DATA_BLOCK "Db Plc <=> HMI"	// DB 100
TITLE = PLC <=> HMI EXCHANGED DATA
AUTHOR : Milesi
VERSION : 0.1
  STRUCT
   BUFFER_DATI : STRUCT
    BD1 : WORD ;	//Numero di ricetta corrente
    BD2 : WORD ;	//Numero di set di dati corrente
    BD3 : WORD ;	//Riservato
    BD4 : WORD ;	//Stato di tresferimento
    BD5 : WORD ;	//Riservato
   END_STRUCT ;
   BUFFER_ORDINI : STRUCT
    BO1 : WORD ;	//0 - Numero di ordine
    BO2 : WORD ;	//Parametro 1
    BO3 : WORD ;	//Parametro 2
    BO4 : WORD ;	//Parametro 3
   END_STRUCT ;
   BUFFER_PAGINE : STRUCT
    BP1 : WORD ;	//Tipo di pagina corrente
    BP2 : WORD ;	//Numero di pagina corrente
    BP3 : WORD ;	//Riservato
    BP4 : WORD ;	//Numero di campo corrente
    BP5 : WORD ;	//Riservato
   END_STRUCT ;
   DB100_DBW28 : WORD ;
   DB100_DBW30 : WORD ;
   DB100_DBW32 : WORD ;
   DB100_DBW34 : WORD ;
   DB100_DBW36 : WORD ;
   DB100_DBW38 : WORD ;
   DB100_DBW40 : WORD ;
   DB100_DBW42 : WORD ;
   DB100_DBW44 : WORD ;
   DB100_DBW46 : WORD ;
   DB100_DBW48 : WORD ;
   DB100_DBW50 : WORD ;
   DB100_DBW52 : WORD ;
   DB100_DBW54 : WORD ;
   DB100_DBW56 : WORD ;
   DB100_DBW58 : WORD ;
   DB100_DBW60 : WORD ;
   DB100_DBW62 : WORD ;
   DB100_DBW64 : WORD ;
   DB100_DBW66 : WORD ;
   DB100_DBW68 : WORD ;
   DB100_DBW70 : WORD ;
   DB100_DBW72 : WORD ;
   DB100_DBW74 : WORD ;
   DB100_DBW76 : WORD ;
   DB100_DBW78 : WORD ;
   DB100_DBW80 : WORD ;
   DB100_DBW82 : WORD ;
   DB100_DBW84 : WORD ;
   DB100_DBW86 : WORD ;
   DB100_DBW88 : WORD ;
   DB100_DBW90 : WORD ;
   DB100_DBW92 : WORD ;
   DB100_DBW94 : WORD ;
   DB100_DBW96 : WORD ;
   DB100_DBW98 : WORD ;
   PROFIBUS : STRUCT
    DB100_DBX100_0 : BOOL ;	//009 Cage 18 motor drive profibus slave 9 fault
    DB100_DBX100_1 : BOOL ;	//010 Cage 12 preforming motor drive profibus slave 10 fault
    DB100_DBX100_2 : BOOL ;	//011 Cage 12 motor drive profibus slave 11 fault
    DB100_DBX100_3 : BOOL ;	//012 Cage 6 motor drive profibus slave 12 fault
    DB100_DBX100_4 : BOOL ;	//013 Take-up unit ET200S profibus slave 20 fault
    DB100_DBX100_5 : BOOL ;	//014 Cage 24 ET200M profibus slave 21 fault
    DB100_DBX100_6 : BOOL ;	//015 Cage 18 ET200M profibus slave 22 fault
    DB100_DBX100_7 : BOOL ;	//016 Cage 12 ET200M profibus slave 23 fault
    DB100_DBX101_0 : BOOL ;	//001 Take-up traverse motor drive profibus slave 3 fault
    DB100_DBX101_1 : BOOL ;	//002 Take-up bobbin motor drive profibus slave 4 fault
    DB100_DBX101_2 : BOOL ;	//003 Capstan motor drive profibus slave 5 fault
    DB100_DBX101_3 : BOOL ;	//004
    DB100_DBX101_4 : BOOL ;	//005
    DB100_DBX101_5 : BOOL ;	//006 Cage 24 preforming motor drive profibus slave 7 fault
    DB100_DBX101_6 : BOOL ;	//007 Cage 24 motor drive profibus slave 6 fault
    DB100_DBX101_7 : BOOL ;	//008 Cage 18 preforming motor drive profibus slave 8 fault
   END_STRUCT ;
   PROFIBUS_1 : STRUCT
    DB100_DBX102_0 : BOOL ;	//025
    DB100_DBX102_1 : BOOL ;	//026
    DB100_DBX102_2 : BOOL ;	//027
    DB100_DBX102_3 : BOOL ;	//028
    DB100_DBX102_4 : BOOL ;	//029
    DB100_DBX102_5 : BOOL ;	//030
    DB100_DBX102_6 : BOOL ;	//031
    DB100_DBX102_7 : BOOL ;	//032
    DB100_DBX103_0 : BOOL ;	//017 Cage 6 ET200M profibus slave 24 fault
    DB100_DBX103_1 : BOOL ;	//018 Pay-off unit ET200S profibus slave 25 fault
    DB100_DBX103_2 : BOOL ;	//019 Pay-off traverse motor drive profibus slave 13 fault
    DB100_DBX103_3 : BOOL ;	//020
    DB100_DBX103_4 : BOOL ;	//021
    DB100_DBX103_5 : BOOL ;	//022
    DB100_DBX103_6 : BOOL ;	//023
    DB100_DBX103_7 : BOOL ;	//024
   END_STRUCT ;
   TRAVERSE : STRUCT
    DB100_DBX104_0 : BOOL ;	//041
    DB100_DBX104_1 : BOOL ;	//042
    DB100_DBX104_2 : BOOL ;	//043
    DB100_DBX104_3 : BOOL ;	//044
    DB100_DBX104_4 : BOOL ;	//045
    DB100_DBX104_5 : BOOL ;	//046
    DB100_DBX104_6 : BOOL ;	//047
    DB100_DBX104_7 : BOOL ;	//048
    DB100_DBX105_0 : BOOL ;	//033 Take-up traverse driven pintle emergency alarm
    DB100_DBX105_1 : BOOL ;	//034 Take-up traverse idle pintle emergency alarm
    DB100_DBX105_2 : BOOL ;	//034 Take-up traverse motor blower overload
    DB100_DBX105_3 : BOOL ;	//036 Take-up traverse motor drive fault
    DB100_DBX105_4 : BOOL ;	//037
    DB100_DBX105_5 : BOOL ;	//038
    DB100_DBX105_6 : BOOL ;	//039
    DB100_DBX105_7 : BOOL ;	//040
   END_STRUCT ;
   TAKE_UP_1 : STRUCT
    DB100_DBX106_0 : BOOL ;	//057 Take-up bobbin down
    DB100_DBX106_1 : BOOL ;	//058 Take-up bobbin off
    DB100_DBX106_2 : BOOL ;	//059
    DB100_DBX106_3 : BOOL ;	//060
    DB100_DBX106_4 : BOOL ;	//061
    DB100_DBX106_5 : BOOL ;	//062
    DB100_DBX106_6 : BOOL ;	//063
    DB100_DBX106_7 : BOOL ;	//064
    DB100_DBX107_0 : BOOL ;	//049 Take-up 24VDC power supply overload
    DB100_DBX107_1 : BOOL ;	//050 Take-up 230VAC power supply overload
    DB100_DBX107_2 : BOOL ;	//051 Take-up AC motors overload
    DB100_DBX107_3 : BOOL ;	//052 Take-up bobbin motor blower overload
    DB100_DBX107_4 : BOOL ;	//053 Take-up bobbin motor electric brake overload
    DB100_DBX107_5 : BOOL ;	//054 Take-up bobbin motor overtemperature
    DB100_DBX107_6 : BOOL ;	//055 Take-up bobbin motor drive fault
    DB100_DBX107_7 : BOOL ;	//056 Take-up bobbin stop series push-button alarm
   END_STRUCT ;
   CAPSTAN : STRUCT
    DB100_DBX108_0 : BOOL ;	//073
    DB100_DBX108_1 : BOOL ;	//074
    DB100_DBX108_2 : BOOL ;	//075
    DB100_DBX108_3 : BOOL ;	//076
    DB100_DBX108_4 : BOOL ;	//077
    DB100_DBX108_5 : BOOL ;	//078
    DB100_DBX108_6 : BOOL ;	//079
    DB100_DBX108_7 : BOOL ;	//080
    DB100_DBX109_0 : BOOL ;	//065 Capstan motor blower overload
    DB100_DBX109_1 : BOOL ;	//066
    DB100_DBX109_2 : BOOL ;	//067 Capstan motor brake control alarm
    DB100_DBX109_3 : BOOL ;	//068 Capstan main air minimum pressure
    DB100_DBX109_4 : BOOL ;	//069 Cable block open alarm
    DB100_DBX109_5 : BOOL ;	//070 Cable block close after run alarm
    DB100_DBX109_6 : BOOL ;	//071 Capstan motor drive fault
    DB100_DBX109_7 : BOOL ;	//072 Capstan motor overtemperature
   END_STRUCT ;
   Spare : STRUCT
    DB100_DBX110_0 : BOOL ;	//089
    DB100_DBX110_1 : BOOL ;	//090
    DB100_DBX110_2 : BOOL ;	//091
    DB100_DBX110_3 : BOOL ;	//092
    DB100_DBX110_4 : BOOL ;	//093
    DB100_DBX110_5 : BOOL ;	//094
    DB100_DBX110_6 : BOOL ;	//095
    DB100_DBX110_7 : BOOL ;	//096
    DB100_DBX111_0 : BOOL ;	//081
    DB100_DBX111_1 : BOOL ;	//082
    DB100_DBX111_2 : BOOL ;	//083
    DB100_DBX111_3 : BOOL ;	//084
    DB100_DBX111_4 : BOOL ;	//085
    DB100_DBX111_5 : BOOL ;	//086
    DB100_DBX111_6 : BOOL ;	//087
    DB100_DBX111_7 : BOOL ;	//088
   END_STRUCT ;
   CAGE24_1 : STRUCT
    DB100_DBX112_00 : BOOL ;	//105 Cage 24 open front guard
    DB100_DBX112_01 : BOOL ;	//106 Cage 24 presence of man
    DB100_DBX112_02 : BOOL ;	//107 Cage 24 loading engaged
    DB100_DBX112_03 : BOOL ;	//108 Cage 24 loading gear box not engaged
    DB100_DBX112_04 : BOOL ;	//109 Cage 24 loading motor overload
    DB100_DBX112_05 : BOOL ;	//110 Cage 24 air pipe not in position
    DB100_DBX112_06 : BOOL ;	//111 Cage 24
    DB100_DBX112_07 : BOOL ;	//112 Cage 24 piston inside cage
    DB100_DBX113_00 : BOOL ;	//097 Cage 24 24VDC power supply overload
    DB100_DBX113_01 : BOOL ;	//098 Cage 24 230VAC power supply overload
    DB100_DBX113_02 : BOOL ;	//099 Cage 24 motor blower overload
    DB100_DBX113_03 : BOOL ;	//100 Cage 24
    DB100_DBX113_04 : BOOL ;	//101 Cage 24 loading platform overload
    DB100_DBX113_05 : BOOL ;	//102 Cage 24 guard blower motor overload
    DB100_DBX113_06 : BOOL ;	//103 Cage 24 open front door
    DB100_DBX113_07 : BOOL ;	//104 Cage 24 open rear door
   END_STRUCT ;
   CAGE24_2 : STRUCT
    DB100_DBX114_00 : BOOL ;	//121 Cage 24 bobbin 1 break of wire
    DB100_DBX114_01 : BOOL ;	//122 Cage 24 bobbin 2 break of wire
    DB100_DBX114_02 : BOOL ;	//123 Cage 24 bobbin 3 break of wire
    DB100_DBX114_03 : BOOL ;	//124 Cage 24 bobbin 4 break of wire
    DB100_DBX114_04 : BOOL ;	//125 Cage 24 bobbin 5 break of wire
    DB100_DBX114_05 : BOOL ;	//126 Cage 24 bobbin 6 break of wire
    DB100_DBX114_06 : BOOL ;	//127 Cage 24 bobbin 7 break of wire
    DB100_DBX114_07 : BOOL ;	//128 Cage 24 bobbin 8 break of wire
    DB100_DBX115_00 : BOOL ;	//113 Cage 24 bobbin 9 break of wire
    DB100_DBX115_01 : BOOL ;	//114 Cage 24 bobbin 10 break of wire
    DB100_DBX115_02 : BOOL ;	//115 Cage 24 bobbin 11 break of wire
    DB100_DBX115_03 : BOOL ;	//116 Cage 24 bobbin 12 break of wire
    DB100_DBX115_04 : BOOL ;	//117 Cage 24 bobbin 13 break of wire
    DB100_DBX115_05 : BOOL ;	//118 Cage 24 bobbin 14 break of wire
    DB100_DBX115_06 : BOOL ;	//119 Cage 24 bobbin 15 break of wire
    DB100_DBX115_07 : BOOL ;	//120 Cage 24 bobbin 16 break of wire
   END_STRUCT ;
   CAGE24_3 : STRUCT
    DB100_DBX116_00 : BOOL ;	//137 Cage 24 bobbin 17 break of wire
    DB100_DBX116_01 : BOOL ;	//138 Cage 24 bobbin 18 break of wire
    DB100_DBX116_02 : BOOL ;	//139 Cage 24 bobbin 19 break of wire
    DB100_DBX116_03 : BOOL ;	//140 Cage 24 bobbin 20 break of wire
    DB100_DBX116_04 : BOOL ;	//141 Cage 24 bobbin 21 break of wire
    DB100_DBX116_05 : BOOL ;	//142 Cage 24 bobbin 22 break of wire
    DB100_DBX116_06 : BOOL ;	//143 Cage 24 bobbin 23 break of wire
    DB100_DBX116_07 : BOOL ;	//144 Cage 24 bobbin 24 break of wire
    DB100_DBX117_00 : BOOL ;	//129
    DB100_DBX117_01 : BOOL ;	//130
    DB100_DBX117_02 : BOOL ;	//131
    DB100_DBX117_03 : BOOL ;	//132
    DB100_DBX117_04 : BOOL ;	//133
    DB100_DBX117_05 : BOOL ;	//134
    DB100_DBX117_06 : BOOL ;	//135 Cage 24 break wire from ring
    DB100_DBX117_07 : BOOL ;	//136 Cage 24 insert wire control alarm
   END_STRUCT ;
   CAGE24_4 : STRUCT
    DB100_DBX118_00 : BOOL ;	//153 Cage 24 main air minumun pressure
    DB100_DBX118_01 : BOOL ;	//154 Cage 24 bobbin brake air tank minimun pressure
    DB100_DBX118_02 : BOOL ;	//155 Cage 24 line 1 open pintles
    DB100_DBX118_03 : BOOL ;	//156 Cage 24 line 2 open pintles
    DB100_DBX118_04 : BOOL ;	//157 Cage 24 line 3 open pintles
    DB100_DBX118_05 : BOOL ;	//158 Cage 24 motor drive fault
    DB100_DBX118_06 : BOOL ;	//159 Cage 24 motor overtemperature
    DB100_DBX118_07 : BOOL ;	//160 Cage 24 Overspeed
    DB100_DBX119_00 : BOOL ;	//145 Cage 24 brakes control alarm
    DB100_DBX119_01 : BOOL ;	//146 Cage 24 platform up
    DB100_DBX119_02 : BOOL ;	//147 Cage 24 Hydraulic unit minimun oil level
    DB100_DBX119_03 : BOOL ;	//148
    DB100_DBX119_04 : BOOL ;	//149 Cage 24 preforming motor electric brake overload
    DB100_DBX119_05 : BOOL ;	//150 Cage 24 preforming motor blower overload
    DB100_DBX119_06 : BOOL ;	//151 Cage 24 preforming open guard
    DB100_DBX119_07 : BOOL ;	//152 Cage 24 preforming motor drive fault
   END_STRUCT ;
   CAGE18_1 : STRUCT
    DB100_DBX120_00 : BOOL ;	//169 Cage 18 open front guard
    DB100_DBX120_01 : BOOL ;	//170 Cage 18 presence of man
    DB100_DBX120_02 : BOOL ;	//171 Cage 18 loading engaged
    DB100_DBX120_03 : BOOL ;	//172 Cage 18 loading gear box not engaged
    DB100_DBX120_04 : BOOL ;	//173 Cage 18 loading motor overload
    DB100_DBX120_05 : BOOL ;	//174 Cage 18 air pipe not in position
    DB100_DBX120_06 : BOOL ;	//175
    DB100_DBX120_07 : BOOL ;	//176 Cage 18 piston inside cage
    DB100_DBX121_00 : BOOL ;	//161 Cage 18 24VDC power supply overload
    DB100_DBX121_01 : BOOL ;	//162 Cage 18 230VAC power supply overload
    DB100_DBX121_02 : BOOL ;	//163 Cage 18 motor blower overload
    DB100_DBX121_03 : BOOL ;	//164
    DB100_DBX121_04 : BOOL ;	//165 Cage 18 loading platform overload
    DB100_DBX121_05 : BOOL ;	//166 Cage 18 guard blower motor overload
    DB100_DBX121_06 : BOOL ;	//167 Cage 18 open front door
    DB100_DBX121_07 : BOOL ;	//168 Cage 18 open rear door
   END_STRUCT ;
   CAGE18_2 : STRUCT
    DB100_DBX122_00 : BOOL ;	//185 Cage 18 bobbin 1 break of wire
    DB100_DBX122_01 : BOOL ;	//186 Cage 18 bobbin 2 break of wire
    DB100_DBX122_02 : BOOL ;	//187 Cage 18 bobbin 3 break of wire
    DB100_DBX122_03 : BOOL ;	//188 Cage 18 bobbin 4 break of wire
    DB100_DBX122_04 : BOOL ;	//189 Cage 18 bobbin 5 break of wire
    DB100_DBX122_05 : BOOL ;	//190 Cage 18 bobbin 6 break of wire
    DB100_DBX122_06 : BOOL ;	//191 Cage 18 bobbin 7 break of wire
    DB100_DBX122_07 : BOOL ;	//192 Cage 18 bobbin 8 break of wire
    DB100_DBX123_00 : BOOL ;	//177 Cage 18 bobbin 9 break of wire
    DB100_DBX123_01 : BOOL ;	//178 Cage 18 bobbin 10 break of wire
    DB100_DBX123_02 : BOOL ;	//179 Cage 18 bobbin 11 break of wire
    DB100_DBX123_03 : BOOL ;	//180 Cage 18 bobbin 12 break of wire
    DB100_DBX123_04 : BOOL ;	//181 Cage 18 bobbin 13 break of wire
    DB100_DBX123_05 : BOOL ;	//182 Cage 18 bobbin 14 break of wire
    DB100_DBX123_06 : BOOL ;	//183 Cage 18 bobbin 15 break of wire
    DB100_DBX123_07 : BOOL ;	//184 Cage 18 bobbin 16 break of wire
   END_STRUCT ;
   CAGE18_3 : STRUCT
    DB100_DBX124_00 : BOOL ;	//201 Cage 18 bobbin 17 break of wire
    DB100_DBX124_01 : BOOL ;	//202 Cage 18 bobbin 18 break of wire
    DB100_DBX124_02 : BOOL ;	//203
    DB100_DBX124_03 : BOOL ;	//204
    DB100_DBX124_04 : BOOL ;	//205
    DB100_DBX124_05 : BOOL ;	//206
    DB100_DBX124_06 : BOOL ;	//207
    DB100_DBX124_07 : BOOL ;	//208
    DB100_DBX125_00 : BOOL ;	//193
    DB100_DBX125_01 : BOOL ;	//194
    DB100_DBX125_02 : BOOL ;	//195
    DB100_DBX125_03 : BOOL ;	//196
    DB100_DBX125_04 : BOOL ;	//197
    DB100_DBX125_05 : BOOL ;	//198
    DB100_DBX125_06 : BOOL ;	//199 Cage 18 break wire from ring
    DB100_DBX125_07 : BOOL ;	//200 Cage 18 insert wire control alarm
   END_STRUCT ;
   CAGE18_4 : STRUCT
    DB100_DBX126_00 : BOOL ;	//217 Cage 18 main air minumun pressure
    DB100_DBX126_01 : BOOL ;	//218 Cage 18 bobbin brake air tank minimun pressure
    DB100_DBX126_02 : BOOL ;	//219 Cage 18 line 1 open pintles
    DB100_DBX126_03 : BOOL ;	//220 Cage 18 line 2 open pintles
    DB100_DBX126_04 : BOOL ;	//221 Cage 18 line 3 open pintles
    DB100_DBX126_05 : BOOL ;	//222 Cage 18 motor drive fault
    DB100_DBX126_06 : BOOL ;	//223 Cage 18 motor overtemperature
    DB100_DBX126_07 : BOOL ;	//224 Cage 18 Overspeed
    DB100_DBX127_00 : BOOL ;	//209 Cage 18 brakes control alarm
    DB100_DBX127_01 : BOOL ;	//210 Cage 18 platform up
    DB100_DBX127_02 : BOOL ;	//211 Cage 18 Hydraulic unit minimun oil level
    DB100_DBX127_03 : BOOL ;	//212 Cage 18
    DB100_DBX127_04 : BOOL ;	//213 Cage 18 preforming motor electric brake overload
    DB100_DBX127_05 : BOOL ;	//214 Cage 18 preforming motor blower overload
    DB100_DBX127_06 : BOOL ;	//215 Cage 18 preforming open guard
    DB100_DBX127_07 : BOOL ;	//216 Cage 18 preforming motor drive fault
   END_STRUCT ;
   CAGE12_1 : STRUCT
    DB100_DBX128_00 : BOOL ;	//233 Cage 12 open front guard
    DB100_DBX128_01 : BOOL ;	//234 Cage 12 presence of man
    DB100_DBX128_02 : BOOL ;	//235 Cage 12 loading engaged
    DB100_DBX128_03 : BOOL ;	//236 Cage 12 loading gear box not engaged
    DB100_DBX128_04 : BOOL ;	//237
    DB100_DBX128_05 : BOOL ;	//238 Cage 12 air pipe not in position
    DB100_DBX128_06 : BOOL ;	//239 Cage 12 loading motor overload
    DB100_DBX128_07 : BOOL ;	//240 Cage 12 piston inside cage
    DB100_DBX129_00 : BOOL ;	//225 Cage 12 24VDC power supply overload
    DB100_DBX129_01 : BOOL ;	//226 Cage 12 230VAC power supply overload
    DB100_DBX129_02 : BOOL ;	//227 Cage 12 motor blower overload
    DB100_DBX129_03 : BOOL ;	//228 Cage 12
    DB100_DBX129_04 : BOOL ;	//229 Cage 12 loading platform overload
    DB100_DBX129_05 : BOOL ;	//230 Cage 12 guard blower motor overload
    DB100_DBX129_06 : BOOL ;	//231 Cage 12 open front door
    DB100_DBX129_07 : BOOL ;	//232 Cage 12 open rear door
   END_STRUCT ;
   Cage12_2 : STRUCT
    DB100_DBX130_00 : BOOL ;	//249 Cage 12 bobbin 1 break of wire
    DB100_DBX130_01 : BOOL ;	//250 Cage 12 bobbin 2 break of wire
    DB100_DBX130_02 : BOOL ;	//251 Cage 12 bobbin 3 break of wire
    DB100_DBX130_03 : BOOL ;	//252 Cage 12 bobbin 4 break of wire
    DB100_DBX130_04 : BOOL ;	//253 Cage 12 bobbin 5 break of wire
    DB100_DBX130_05 : BOOL ;	//254 Cage 12 bobbin 6 break of wire
    DB100_DBX130_06 : BOOL ;	//255 Cage 12 bobbin 7 break of wire
    DB100_DBX130_07 : BOOL ;	//256 Cage 12 bobbin 8 break of wire
    DB100_DBX131_00 : BOOL ;	//241 Cage 12 bobbin 9 break of wire
    DB100_DBX131_01 : BOOL ;	//242 Cage 12 bobbin 10 break of wire
    DB100_DBX131_02 : BOOL ;	//243 Cage 12 bobbin 11 break of wire
    DB100_DBX131_03 : BOOL ;	//244 Cage 12 bobbin 12 break of wire
    DB100_DBX131_04 : BOOL ;	//245
    DB100_DBX131_05 : BOOL ;	//246
    DB100_DBX131_06 : BOOL ;	//247
    DB100_DBX131_07 : BOOL ;	//248
   END_STRUCT ;
   Cage12_3 : STRUCT
    DB100_DBX132_00 : BOOL ;	//265 Cage 12
    DB100_DBX132_01 : BOOL ;	//266 Cage 12
    DB100_DBX132_02 : BOOL ;	//267 Cage 12
    DB100_DBX132_03 : BOOL ;	//268 Cage 12
    DB100_DBX132_04 : BOOL ;	//269 Cage 12
    DB100_DBX132_05 : BOOL ;	//270 Cage 12
    DB100_DBX132_06 : BOOL ;	//271 Cage 12
    DB100_DBX132_07 : BOOL ;	//272 Cage 12
    DB100_DBX133_00 : BOOL ;	//257 Cage 12
    DB100_DBX133_01 : BOOL ;	//258 Cage 12
    DB100_DBX133_02 : BOOL ;	//259 Cage 12
    DB100_DBX133_03 : BOOL ;	//260 Cage 12
    DB100_DBX133_04 : BOOL ;	//261 Cage 12
    DB100_DBX133_05 : BOOL ;	//262 Cage 12
    DB100_DBX133_06 : BOOL ;	//263 Cage 12 break wire from ring
    DB100_DBX133_07 : BOOL ;	//264 Cage 12 insert wire control alarm
   END_STRUCT ;
   Cage12_4 : STRUCT
    DB100_DBX134_00 : BOOL ;	//281 Cage 12 main air minumun pressure
    DB100_DBX134_01 : BOOL ;	//282 Cage 12 bobbin brake air tank minimun pressure
    DB100_DBX134_02 : BOOL ;	//283 Cage 12 line 1 open pintles
    DB100_DBX134_03 : BOOL ;	//284 Cage 12 line 2 open pintles
    DB100_DBX134_04 : BOOL ;	//285 Cage 12 line 3 open pintles
    DB100_DBX134_05 : BOOL ;	//286 Cage 12 motor drive fault
    DB100_DBX134_06 : BOOL ;	//287 Cage 12 motor overtemperature
    DB100_DBX134_07 : BOOL ;	//288 Cage 12 Overspeed
    DB100_DBX135_00 : BOOL ;	//273 Cage 12 brakes control alarm
    DB100_DBX135_01 : BOOL ;	//274 Cage 12 platform up
    DB100_DBX135_02 : BOOL ;	//275 Cage 12 Hydraulic unit minimun oil level
    DB100_DBX135_03 : BOOL ;	//276 Cage 12
    DB100_DBX135_04 : BOOL ;	//277 Cage 12 preforming motor electric brake overload
    DB100_DBX135_05 : BOOL ;	//278 Cage 12 preforming motor blower overload
    DB100_DBX135_06 : BOOL ;	//279 Cage 12 preforming open guard
    DB100_DBX135_07 : BOOL ;	//280 Cage 12 preforming motor drive fault
   END_STRUCT ;
   Cage6_1 : STRUCT
    DB100_DBX136_0 : BOOL ;	//297 Cage 6 open front guard
    DB100_DBX136_1 : BOOL ;	//298 Cage 6 presence of man
    DB100_DBX136_2 : BOOL ;	//299 Cage 6 loading engaged
    DB100_DBX136_3 : BOOL ;	//300 Cage 6 loading gear box not engaged
    DB100_DBX136_4 : BOOL ;	//301 Cage 6
    DB100_DBX136_5 : BOOL ;	//302 Cage 6 air pipe not in position
    DB100_DBX136_6 : BOOL ;	//303 Cage 6 loading motor overload
    DB100_DBX136_7 : BOOL ;	//304 Cage 6 piston inside cage
    DB100_DBX137_0 : BOOL ;	//289 Cage 6 24VDC power supply overload
    DB100_DBX137_1 : BOOL ;	//290 Cage 6 230VAC power supply overload
    DB100_DBX137_2 : BOOL ;	//291 Cage 6 motor blower overload
    DB100_DBX137_3 : BOOL ;	//292 Cage 6
    DB100_DBX137_4 : BOOL ;	//293 Cage 6 loading platform overload
    DB100_DBX137_5 : BOOL ;	//294 Cage 6 guard blower motor overload
    DB100_DBX137_6 : BOOL ;	//295 Cage 6 open front door
    DB100_DBX137_7 : BOOL ;	//296 Cage 6 open rear door
   END_STRUCT ;
   Cage6_2 : STRUCT
    DB100_DBX138_0 : BOOL ;	//313 Cage 6 bobbin 1 break of wire
    DB100_DBX138_1 : BOOL ;	//314 Cage 6 bobbin 2 break of wire
    DB100_DBX138_2 : BOOL ;	//315 Cage 6 bobbin 3 break of wire
    DB100_DBX138_3 : BOOL ;	//316 Cage 6 bobbin 4 break of wire
    DB100_DBX138_4 : BOOL ;	//317 Cage 6 bobbin 5 break of wire
    DB100_DBX138_5 : BOOL ;	//318 Cage 6 bobbin 6 break of wire
    DB100_DBX138_6 : BOOL ;	//319 Cage 6
    DB100_DBX138_7 : BOOL ;	//320 Cage 6
    DB100_DBX139_0 : BOOL ;	//305 Cage 6
    DB100_DBX139_1 : BOOL ;	//306 Cage 6
    DB100_DBX139_2 : BOOL ;	//307 Cage 6
    DB100_DBX139_3 : BOOL ;	//308 Cage 6
    DB100_DBX139_4 : BOOL ;	//309 Cage 6
    DB100_DBX139_5 : BOOL ;	//310 Cage 6
    DB100_DBX139_6 : BOOL ;	//311 Cage 6
    DB100_DBX139_7 : BOOL ;	//312 Cage 6
   END_STRUCT ;
   Cage6_3 : STRUCT
    DB100_DBX140_0 : BOOL ;	//329 Cage 6
    DB100_DBX140_1 : BOOL ;	//330 Cage 6
    DB100_DBX140_2 : BOOL ;	//331 Cage 6
    DB100_DBX140_3 : BOOL ;	//332 Cage 6
    DB100_DBX140_4 : BOOL ;	//333 Cage 6
    DB100_DBX140_5 : BOOL ;	//334 Cage 6
    DB100_DBX140_6 : BOOL ;	//335 Cage 6
    DB100_DBX140_7 : BOOL ;	//336 Cage 6
    DB100_DBX141_0 : BOOL ;	//321 Cage 6
    DB100_DBX141_1 : BOOL ;	//322 Cage 6
    DB100_DBX141_2 : BOOL ;	//323 Cage 6
    DB100_DBX141_3 : BOOL ;	//324 Cage 6
    DB100_DBX141_4 : BOOL ;	//325 Cage 6
    DB100_DBX141_5 : BOOL ;	//326 Cage 6
    DB100_DBX141_6 : BOOL ;	//327 Cage 6 break wire from ring
    DB100_DBX141_7 : BOOL ;	//328 Cage 6 insert wire control alarm
   END_STRUCT ;
   Cage6_4 : STRUCT
    DB100_DBX142_0 : BOOL ;	//345 Cage 6 main air minumun pressure
    DB100_DBX142_1 : BOOL ;	//346 Cage 6 bobbin brake air tank minimun pressure
    DB100_DBX142_2 : BOOL ;	//347 Cage 6 line 1 open pintles
    DB100_DBX142_3 : BOOL ;	//348 Cage 6 line 2 open pintles
    DB100_DBX142_4 : BOOL ;	//349 Cage 6 line 3 open pintles
    DB100_DBX142_5 : BOOL ;	//350 Cage 6 motor drive fault
    DB100_DBX142_6 : BOOL ;	//351 Cage 6 motor overtemperature
    DB100_DBX142_7 : BOOL ;	//352 Cage 6 Overspeed
    DB100_DBX143_0 : BOOL ;	//337 Cage 6 brakes control alarm
    DB100_DBX143_1 : BOOL ;	//338 Cage 6 platform up
    DB100_DBX143_2 : BOOL ;	//339 Cage 6 Hydraulic unit minimun oil level
    DB100_DBX143_3 : BOOL ;	//340 Cage 6
    DB100_DBX143_4 : BOOL ;	//341 Cage 6
    DB100_DBX143_5 : BOOL ;	//342 Cage 6
    DB100_DBX143_6 : BOOL ;	//343 Cage 6 preforming open guard
    DB100_DBX143_7 : BOOL ;	//344 Cage 6
   END_STRUCT ;
   PAY_OFF_UNIT1 : STRUCT
    DB100_DBX144_0 : BOOL ;	//361 Pay-off traverse driven pintle emergency alarm
    DB100_DBX144_1 : BOOL ;	//362 Pay-off traverse idle pintle emergency alarm
    DB100_DBX144_2 : BOOL ;	//363 Pay-off traverse motor drive fault
    DB100_DBX144_3 : BOOL ;	//364
    DB100_DBX144_4 : BOOL ;	//365
    DB100_DBX144_5 : BOOL ;	//366
    DB100_DBX144_6 : BOOL ;	//367
    DB100_DBX144_7 : BOOL ;	//368
    DB100_DBX145_0 : BOOL ;	//353 Pay-off 24VDC power supply overload
    DB100_DBX145_1 : BOOL ;	//354 Pay-off 230VAC power supply overload
    DB100_DBX145_2 : BOOL ;	//355 Pay-off AC motors overload
    DB100_DBX145_3 : BOOL ;	//356 Pay-off bobbin down
    DB100_DBX145_4 : BOOL ;	//357
    DB100_DBX145_5 : BOOL ;	//358 Pay-off main air minimum pressure
    DB100_DBX145_6 : BOOL ;	//359 Pay-off bobbin break of wire
    DB100_DBX145_7 : BOOL ;	//360 Pay-off traverse motor blower overload
   END_STRUCT ;
   CENTRAL_PAY_OFF : STRUCT
    DB100_DBX146_00 : BOOL ;	//377
    DB100_DBX146_01 : BOOL ;	//378
    DB100_DBX146_02 : BOOL ;	//379
    DB100_DBX146_03 : BOOL ;	//380
    DB100_DBX146_04 : BOOL ;	//381
    DB100_DBX146_05 : BOOL ;	//382
    DB100_DBX146_06 : BOOL ;	//383
    DB100_DBX146_07 : BOOL ;	//384
    DB100_DBX147_00 : BOOL ;	//369 Pay-off 630 open pintles
    DB100_DBX147_01 : BOOL ;	//370 Pay-off 630 break of wire
    DB100_DBX147_02 : BOOL ;	//371 Pay-off 630 main air minimum pressure
    DB100_DBX147_03 : BOOL ;	//372 Pay-off 630 brake off
    DB100_DBX147_04 : BOOL ;	//373
    DB100_DBX147_05 : BOOL ;	//374
    DB100_DBX147_06 : BOOL ;	//375
    DB100_DBX147_07 : BOOL ;	//376
   END_STRUCT ;
   LINE1 : STRUCT
    DB100_DBX148_0 : BOOL ;	//393 Line stop from metercounter alarm
    DB100_DBX148_1 : BOOL ;	//394 AC motor drives feeder DC BUS fault
    DB100_DBX148_2 : BOOL ;	//395 Control desk fan overload
    DB100_DBX148_3 : BOOL ;	//396 Drives auxiliary 110VAC transformer overload
    DB100_DBX148_4 : BOOL ;	//397 Dryer supply overload
    DB100_DBX148_5 : BOOL ;	//398 AC motor drives feeder braking resistor alarm
    DB100_DBX148_6 : BOOL ;	//399 Machine running
    DB100_DBX148_7 : BOOL ;	//400 Ready to run
    DB100_DBX149_0 : BOOL ;	//385 Auxiliary off
    DB100_DBX149_1 : BOOL ;	//386 Emergency push-button alarm
    DB100_DBX149_2 : BOOL ;	//387 Cabinet overtemperature alarm
    DB100_DBX149_3 : BOOL ;	//388 Service auxiliary 230V transformer overload
    DB100_DBX149_4 : BOOL ;	//389 Cabinet air fans overload
    DB100_DBX149_5 : BOOL ;	//390 Line stop series push-button alarm
    DB100_DBX149_6 : BOOL ;	//391 Linear overspeed alarm
    DB100_DBX149_7 : BOOL ;	//392 Line slow-down from metercounter alarm
   END_STRUCT ;
   LINE_21 : STRUCT
    DB100_DBX150_0 : BOOL ;	//409 24DC auxiliary feeding overload
    DB100_DBX150_1 : BOOL ;	//410 230AC auxiliary feeding overload
    DB100_DBX150_2 : BOOL ;	//411 AC motor drive feeder fan overload
    DB100_DBX150_3 : BOOL ;	//412 24DC plc input supply overload
    DB100_DBX150_4 : BOOL ;	//413
    DB100_DBX150_5 : BOOL ;	//414
    DB100_DBX150_6 : BOOL ;	//415
    DB100_DBX150_7 : BOOL ;	//416
    DB100_DBX151_0 : BOOL ;	//401 230AC UPS module alarm
    DB100_DBX151_1 : BOOL ;	//402 230AC UPS battery nearly low
    DB100_DBX151_2 : BOOL ;	//403 230VAC UPS line voltage missing - UPS is operating
    DB100_DBX151_3 : BOOL ;	//404 24DC UPS module alarm
    DB100_DBX151_4 : BOOL ;	//405 24DC UPS line voltage missing - UPS is operating
    DB100_DBX151_5 : BOOL ;	//405
    DB100_DBX151_6 : BOOL ;	//407
    DB100_DBX151_7 : BOOL ;	//408
   END_STRUCT ;
  END_STRUCT ;	
BEGIN
   TAKE_UP_1.DB100_DBX106_1 := TRUE;
   CAGE24_4.DB100_DBX118_00 := TRUE;
   CAGE18_4.DB100_DBX126_00 := TRUE;
   Cage6_4.DB100_DBX142_0 := TRUE;
END_DATA_BLOCK

DATA_BLOCK "Count setting"	// DB 101
TITLE = COUNT SETTINGS DATA BLOCK
AUTHOR : Milesi
VERSION : 0.1
  STRUCT
   DINT0 : DINT ;
   DINT4 : DINT ;
   DINT8 : DINT ;
   DINT12 : DINT ;
  END_STRUCT ;	
BEGIN
   DINT4 := L#16777216;
   DINT8 := L#-61325;
   DINT12 := L#4292608;
END_DATA_BLOCK

DATA_BLOCK "FB125"	// DB 125
TITLE = DB FB125 DATA BLOCK
AUTHOR : SIEMENS
FAMILY : DP
VERSION : 0.0
"DETAIL_DP_DIAG"
BEGIN
END_DATA_BLOCK

ORGANIZATION_BLOCK "Cycle execution"	// OB 1
TITLE = CYCLE EXECUTION ORGANIZATION BLOCK
AUTHOR : Milesi
VERSION : 0.1
VAR_TEMP
  OB1_EV_CLASS : BYTE ;	//Bits 0-3 = 1 (Coming event), Bits 4-7 = 1 (Event class 1)
  OB1_SCAN_1 : BYTE ;	//1 (Cold restart scan 1 of OB 1), 3 (Scan 2-n of OB 1)
  OB1_PRIORITY : BYTE ;	//Priority of OB Execution
  OB1_OB_NUMBR : BYTE ;	//1 (Organization block 1, OB1)
  OB1_RESERVED_1 : BYTE ;	//Reserved for system
  OB1_RESERVED_2 : BYTE ;	//Reserved for system
  OB1_PREV_CYCLE : INT ;	//Cycle time of previous OB1 scan (milliseconds)
  OB1_MIN_CYCLE : INT ;	//Minimum cycle time of OB1 (milliseconds)
  OB1_MAX_CYCLE : INT ;	//Maximum cycle time of OB1 (milliseconds)
  OB1_DATE_TIME : DATE_AND_TIME ;	//Date and time OB1 started
END_VAR
BEGIN
NETWORK
TITLE = ALARMS RESET
      A(;
      O     "MAP_DI".DB91_DBX002_3;
      O     "MAP_DI".DB91_DBX022_3;
      O     "MAP_DI".DB91_DBX042_3;
      O     "MAP_DI".DB91_DBX062_3;
      O     "MAP_DI".DB91_DBX082_3;
      );
      AN    "M180.1";
      =     "M30.1";
      A     "M30.1";
      CC    "Alarms Reset";
NETWORK
TITLE = DRIVES FAULT RESET
      A     "M30.1";
      =     "Plc --> Drives".TRAVERSE_CONTROL_W1.DB2_DBX1_7;
      =     "Plc --> Drives".BOBBIN_CONTROL_W1.DB2_DBX41_7;
      =     "Plc --> Drives".CAPSTAN_CONTROL_W1.DB2_DBX81_7;
      =     "Plc --> Drives".CAGE_24_PREF_CONTROL_W1.DB2_DBX121_7;
      =     "Plc --> Drives".CAGE_24_CONTROL_W1.DB2_DBX161_7;
      =     "Plc --> Drives".CAGE_18_PREF_CONTROL_W1.DB2_DBX201_7;
      =     "Plc --> Drives".CAGE_18_CONTROL_W1.DB2_DBX241_7;
      =     "Plc --> Drives".CAGE_12_PREF_CONTROL_W1.DB2_DBX281_7;
      =     "Plc --> Drives".CAGE_12_CONTROL_W1.DB2_DBX321_7;
      =     "Plc --> Drives".CAGE_6_CONTROL_W1.DB2_DBX361_7;
      =     "MAP_DO".DB93_DBX000_4;
      =     "MAP_DO".DB93_DBX000_5;
NETWORK
TITLE = PROGRAMS CALL
      CALL  "Profibus unit";
      CALL  "Take-up traverse alarms";
      CALL  "Take-up traverse unit";
      CALL  "Take-up alarms";
      CALL  "Take-up unit";
      CALL  "Capstan alarms";
      CALL  "Capstan unit";
      CALL  "Cage common function";
      CALL  "Cage 24 alarms";
      CALL  "Cage 24 unit";
      CALL  "Cage 24 loading fase";
      CALL  "Cage 24 preforming alarm";
      CALL  "Cage 24 preforming unit";
      CALL  "Cage 18 alarms";
      CALL  "Cage 18 unit";
      CALL  "Cage 18 loading fase";
      CALL  "Cage 18 preforming alarm";
      CALL  "Cage 18 preforming unit";
      CALL  "Cage 12 alarms";
      CALL  "Cage 12 unit";
      CALL  "Cage 12 loading fase";
      CALL  "Cage 12 preforming alarm";
      CALL  "Cage 12 preforming unit";
      CALL  "Cage 6 alarms";
      CALL  "Cage 6 unit";
      CALL  "Cage 6 loading fase";
      CALL  "Cage 6 preforming alarms";
      CALL  "Cage 6 preforming unit";
      CALL  "Pay-off 630 alarms";
      CALL  "Pay-off 630 unit";
      CALL  "Metercounter alarms";
      CALL  "Metercounter unit";
      CALL  "Common function";
      CALL  "Hour counter";
      CALL  "Line alarms";
      CALL  "Line unit";
      CALL  "Run consent";
      CALL  "Line jog - line run";
      CALL  "Line reference";
      CALL  "Linear speed";
      CALL  "Missing power supply";
      CALL  "HMI animation unit";
      CALL  "Take-up traverse impulse";
      CALL  "Cage 24 wires insertion";
      CALL  "Cage 18 wires insertion";
      CALL  "Cage 12 wires insertion";
      CALL  "Cage 6 wires insertion";
      CALL  "Wires break time";
      CALL  "Bobbins diameter";
      CALL  "Bobbins brake";
      CALL  "Rpm increase";
      CALL  "Map Input Function";
      CALL  "Map Output Function";
NETWORK
TITLE = PROFIBUS DIAGNOSTIC
      CALL  "DETAIL_DP_DIAG" , "FB125" (
           DIW 0                    := 1,
           DIX 2.0                  := FALSE,
           DIX 2.2                  := "M1.5",
           DIB 6                    := "MB304");
END_ORGANIZATION_BLOCK

ORGANIZATION_BLOCK "Diagnostic interrupt"	// OB 82
TITLE = DIAGNOSTIC INTERRUPT ORGANIZATION BLOCK
AUTHOR : Milesi
VERSION : 0.1
VAR_TEMP
  OB82_EV_CLASS : BYTE ;	//16#39, Event class 3, Entering event state, Internal fault event
  OB82_FLT_ID : BYTE ;	//16#XX, Fault identifcation code
  OB82_PRIORITY : BYTE ;	//Priority of OB Execution
  OB82_OB_NUMBR : BYTE ;	//82 (Organization block 82, OB82)
  OB82_RESERVED_1 : BYTE ;	//Reserved for system
  OB82_IO_FLAG : BYTE ;	//Input (01010100), Output (01010101)
  OB82_MDL_ADDR : WORD ;	//Base address of module with fault
  OB82_MDL_DEFECT : BOOL ;	//Module defective
  OB82_INT_FAULT : BOOL ;	//Internal fault
  OB82_EXT_FAULT : BOOL ;	//External fault
  OB82_PNT_INFO : BOOL ;	//Point information
  OB82_EXT_VOLTAGE : BOOL ;	//External voltage low
  OB82_FLD_CONNCTR : BOOL ;	//Field wiring connector missing
  OB82_NO_CONFIG : BOOL ;	//Module has no configuration data
  OB82_CONFIG_ERR : BOOL ;	//Module has configuration error
  OB82_MDL_TYPE : BYTE ;	//Type of module
  OB82_SUB_MDL_ERR : BOOL ;	//Sub-Module is missing or has error
  OB82_COMM_FAULT : BOOL ;	//Communication fault
  OB82_MDL_STOP : BOOL ;	//Module is stopped
  OB82_WTCH_DOG_FLT : BOOL ;	//Watch dog timer stopped module
  OB82_INT_PS_FLT : BOOL ;	//Internal power supply fault
  OB82_PRIM_BATT_FLT : BOOL ;	//Primary battery is in fault
  OB82_BCKUP_BATT_FLT : BOOL ;	//Backup battery is in fault
  OB82_RESERVED_2 : BOOL ;	//Reserved for system
  OB82_RACK_FLT : BOOL ;	//Rack fault, only for bus interface module
  OB82_PROC_FLT : BOOL ;	//Processor fault
  OB82_EPROM_FLT : BOOL ;	//EPROM fault
  OB82_RAM_FLT : BOOL ;	//RAM fault
  OB82_ADU_FLT : BOOL ;	//ADU fault
  OB82_FUSE_FLT : BOOL ;	//Fuse fault
  OB82_HW_INTR_FLT : BOOL ;	//Hardware interupt input in fault
  OB82_RESERVED_3 : BOOL ;	//Reserved for system
  OB82_DATE_TIME : DATE_AND_TIME ;	//Date and time OB82 started
END_VAR
BEGIN
NETWORK
TITLE = PROFIBUS DIAGNOSTIC
      CALL  "DETAIL_DP_DIAG" , "FB125" (
           DIW 0                    := 1,
           DIX 2.0                  := FALSE,
           DIX 2.2                  := "M1.5",
           DIB 6                    := "MB304");
END_ORGANIZATION_BLOCK

ORGANIZATION_BLOCK "Rack failure"	// OB 86
TITLE = RACK FAILURE ORGANIZATION BLOCK
AUTHOR : Milesi
VERSION : 0.1
VAR_TEMP
  OB86_EV_CLASS : BYTE ;	//16#38/39 Event class 3
  OB86_FLT_ID : BYTE ;	//16#C1/C4/C5, Fault identifcation code
  OB86_PRIORITY : BYTE ;	//Priority of OB Execution
  OB86_OB_NUMBR : BYTE ;	//86 (Organization block 86, OB86)
  OB86_RESERVED_1 : BYTE ;	//Reserved for system
  OB86_RESERVED_2 : BYTE ;	//Reserved for system
  OB86_MDL_ADDR : INT ;	//Base address of IM module in rack with fault
  OB86_RACKS_FLTD : ARRAY  [0 .. 31 ] OF BOOL ;	//Racks in fault
  OB86_DATE_TIME : DATE_AND_TIME ;	//Date and time OB86 started
END_VAR
BEGIN
NETWORK
TITLE = PROFIBUS DIAGNOSTIC
      CALL  "DETAIL_DP_DIAG" , "FB125" (
           DIW 0                    := 1,
           DIX 2.0                  := FALSE,
           DIX 2.2                  := "M1.5",
           DIB 6                    := "MB304");
END_ORGANIZATION_BLOCK

ORGANIZATION_BLOCK "Startup"	// OB 100
TITLE = STARTUP ORGANIZATION BLOCK
AUTHOR : Milesi
VERSION : 0.1
VAR_TEMP
  OB100_EV_CLASS : BYTE ;	//16#13, Event class 1, Entering event state, Event logged in diagnostic buffer
  OB100_STRTUP : BYTE ;	//16#81/82/83/84 Method of startup
  OB100_PRIORITY : BYTE ;	//27 (Priority of 1 is lowest)
  OB100_OB_NUMBR : BYTE ;	//100 (Organization block 100, OB100)
  OB100_RESERVED_1 : BYTE ;	//Reserved for system
  OB100_RESERVED_2 : BYTE ;	//Reserved for system
  OB100_STOP : WORD ;	//Event that caused CPU to stop (16#4xxx)
  OB100_STRT_INFO : DWORD ;	//Information on how system started
  OB100_DATE_TIME : DATE_AND_TIME ;	//Date and time OB100 started
END_VAR
BEGIN
NETWORK
TITLE = 6SE70 DRIVES CONTROL WORD 1 RESET
      L     W#16#404;
      T     "Plc --> Drives".TRAVERSE_CONTROL_W1;
      T     "Plc --> Drives".BOBBIN_CONTROL_W1;
      T     "Plc --> Drives".CAPSTAN_CONTROL_W1;
      T     "Plc --> Drives".CAGE_24_PREF_CONTROL_W1;
      T     "Plc --> Drives".CAGE_24_CONTROL_W1;
      T     "Plc --> Drives".CAGE_18_PREF_CONTROL_W1;
      T     "Plc --> Drives".CAGE_18_CONTROL_W1;
      T     "Plc --> Drives".CAGE_12_PREF_CONTROL_W1;
      T     "Plc --> Drives".CAGE_12_CONTROL_W1;
      T     "Plc --> Drives".CAGE_6_CONTROL_W1;
NETWORK
TITLE = 6SE70 DRIVES CONTROL WORD 2 RESET
      L     W#16#0;
      T     "Plc --> Drives".TRAVERSE_CONTROL_W2;
      T     "Plc --> Drives".BOBBIN_CONTROL_W2;
      T     "Plc --> Drives".CAPSTAN_CONTROL_W2;
      T     "Plc --> Drives".CAGE_24_PREF_CONTROL_W2;
      T     "Plc --> Drives".CAGE_24_CONTROL_W2;
      T     "Plc --> Drives".CAGE_18_PREF_CONTROL_W2;
      T     "Plc --> Drives".CAGE_18_CONTROL_W2;
      T     "Plc --> Drives".CAGE_12_PREF_CONTROL_W2;
      T     "Plc --> Drives".CAGE_12_CONTROL_W2;
      T     "Plc --> Drives".CAGE_6_CONTROL_W2;
NETWORK
TITLE = METERCOUNTER RESET
      L     0.000000e+00;
      T     "Take-up traverse".DB5_DBD44;
      T     "Metercounter".DB41_DBD132;
END_ORGANIZATION_BLOCK

ORGANIZATION_BLOCK "MOD_ERR"	// OB 122
TITLE = "Module Access Error"
VERSION : 0.1
VAR_TEMP
  OB122_EV_CLASS : BYTE ;	//16#29, Event class 2, Entering event state, Internal fault event
  OB122_SW_FLT : BYTE ;	//16#XX Software error code
  OB122_PRIORITY : BYTE ;	//Priority of OB Execution
  OB122_OB_NUMBR : BYTE ;	//122 (Organization block 122, OB122)
  OB122_BLK_TYPE : BYTE ;	//16#88/8C/8E Type of block fault occured in
  OB122_MEM_AREA : BYTE ;	//Memory area where access error occured
  OB122_MEM_ADDR : WORD ;	//Memory address where access error occured
  OB122_BLK_NUM : WORD ;	//Block number in which error occured
  OB122_PRG_ADDR : WORD ;	//Program address where error occured
  OB122_DATE_TIME : DATE_AND_TIME ;	//Date and time OB1 started
END_VAR
BEGIN
// (block stored without names or comments; labels and parameter names are numbered)
END_ORGANIZATION_BLOCK

SYMBOL_TABLE
"Cage Function"	FC 7	FC 7	// Cage Function
"Translation Function"	FC 8	FC 8	// Translation Function
"Clamp Function"	FC 9	FC 9	// Clamp Function
"Rotation Function"	FC 10	FC 10	// Rotation Function
"E0.0"	I 0.0	BOOL	// Loader Lifting Push Button - 274S1
"E0.1"	I 0.1	BOOL	// Loader Lowering Push Button - 274S2
"E0.2"	I 0.2	BOOL	// Alarms Reset Push Button - 274S3
"E0.3"	I 0.3	BOOL	// Loader Translation Zero Speed from Drive 251G1
"E0.4"	I 0.4	BOOL	// Loader in position Enabled to LOAD Proximity 274B5
"E0.5"	I 0.5	BOOL	// Loader in position Enabled to UNLOAD Proximity 274B6
"E0.6"	I 0.6	BOOL	// Spare
"E0.7"	I 0.7	BOOL	// Spare
"E1.0"	I 1.0	BOOL	// Loader ENABLE for Stand-By ZONE From MAIN BOARD
"E1.1"	I 1.1	BOOL	// Loader Presence of Bobbin in Cage form MAIN BOARD
"E1.2"	I 1.2	BOOL	// Loader Piston Block Inserted from MAIN BOARD  ?????
"E1.3"	I 1.3	BOOL	// Pintles OPEN from MAIN BOARD
"E1.4"	I 1.4	BOOL	// Spare
"E1.5"	I 1.5	BOOL	// Spare
"E1.6"	I 1.6	BOOL	// Spare
"E1.7"	I 1.7	BOOL	// Spare
"E124.0"	I 124.0	BOOL	// Loader Translation FRONT Limit-Switch - 271S1 - 271S1.1 - [1=.....]
"E124.1"	I 124.1	BOOL	// Loader Translation REAR Limit-Switch - 271S2 - 271S2.2 - [1=......]
"E124.2"	I 124.2	BOOL	// Loader Translation SLOW-DOWN Limit Switch - 271B3 - [1=Slow-Down]
"E124.3"	I 124.3	BOOL	// Loader Inside Cage STOP Translation Sensor - 271B4 - [1=Stop]
"E124.4"	I 124.4	BOOL	// Loader Translation Run FORWARD Push-Button - 271S5 - [1=Run FW]
"E124.5"	I 124.5	BOOL	// Loader Translation Run BACKWARD Push-Button - 271S6 - [1=Run BW]
"E124.6"	I 124.6	BOOL	// Loader Translation Slow Run Forward-PB - 271S7 - [1=Run FW]
"E124.7"	I 124.7	BOOL	// Loader Translation Slow Run Backward-PB - 271S8 - [1=Run BW]
"E125.0"	I 125.0	BOOL	// Loader Bobbins Lift / Lower Drives  Fault - 252G1 - 253G1 - 246Q2 - [0=Fault]
"E125.1"	I 125.1	BOOL	// Loader Bobbins UP Limit-Switch - 272S2 - [1=Up]
"E125.2"	I 125.2	BOOL	// Loader Bobbins DOWN Limit-Switch - 272S3 - [1=Down]
"E125.3"	I 125.3	BOOL	// Spare
"E125.4"	I 125.4	BOOL	// Loader Bobbins Presence ON Loader - 272B5 - [1=On]
"E125.5"	I 125.5	BOOL	// Loader Bobbins Presence UNDER Loader - 272B6 - [1=Under]
"E125.6"	I 125.6	BOOL	// Loader Translation STAND-BY Sensor 272S7 - [1=Stand-By]
"E125.7"	I 125.7	BOOL	// Loader Bobbin At Rest Back Limit-Switch - 272S8 - [1=.....]
"E126.0"	I 126.0	BOOL	// Auxiliary Circuits ON - 242K1 - [1=ON]
"E126.1"	I 126.1	BOOL	// Cabinet Fan Overload - 245Q1 - [0=Overload]
"E126.2"	I 126.2	BOOL	// Loader Clamp OPEN / CLOSE Motor Overload - 244Q1 - [1=Overload]
"E126.3"	I 126.3	BOOL	// Loader Clamp OPEN Limit Switch - 273S2 - [1=Open]
"E126.4"	I 126.4	BOOL	// Loader Clamp CLOSE Limit Switch - 273S3 - [1=Close]
"E126.5"	I 126.5	BOOL	// Loader Clamp OPEN Push-Button - 271S5 - [1=Open]
"E126.6"	I 126.6	BOOL	// Loader Clamp CLOSE Push-Button - 271S6 - [1=Close]
"E126.7"	I 126.7	BOOL	// Loader Translation FAULT - 252G1 - 246Q3 - 246Q1 - 251F2 - 251F3 - [0=Fault]
"M0.0"	M 0.0	BOOL	// Bit Always OFF
"M0.1"	M 0.1	BOOL	// Bit Always ON
"M1.5"	M 1.5	BOOL	// Merker clock 1sec.
"M3.0"	M 3.0	BOOL	// Enable to move searching loading position
"M3.1"	M 3.1	BOOL	// Enable to move searching unloading position
"M4.0"	M 4.0	BOOL	// FP Enable to move Forward
"M4.1"	M 4.1	BOOL	// FP Enable to move Backward
"m6.0"	M 6.0	BOOL	// No slow down forward direction
"M6.1"	M 6.1	BOOL	// No slow down ackward directon
"M8.0"	M 8.0	BOOL	// Loader inside cage - stop forward translation
"M10.0"	M 10.0	BOOL	// Stop bit FORWARD
"M10.1"	M 10.1	BOOL	// Stop bit FORWARD One-Shot
"M010.2"	M 10.2	BOOL	// Backward stop bit
"M10.4"	M 10.4	BOOL	// Loader UP Consent bit
"M10.5"	M 10.5	BOOL	// Loader DOWN Consent Bit
"M10.6"	M 10.6	BOOL	// Loader UP Enable
"M10.7"	M 10.7	BOOL	// Loader DOWN Enable
"M12.0"	M 12.0	BOOL	// Slow-Down Stand-by Zone
"M13.0"	M 13.0	BOOL	// Bobbin not in loader
"m13.3"	M 13.3	BOOL	// Loader in stand-by zone slow down bit
"M15.1"	M 15.1	BOOL	// Loader consent bit in Cage FORWARD
"M15.2"	M 15.2	BOOL	// Loader consent bit in Cage BACKWARD
"M15.3"	M 15.3	BOOL	// LOADER ENABLE FORWARD IN CAGE
"M17.0"	M 17.0	BOOL	// Translation consent
"M17.1"	M 17.1	BOOL	// Loader FORWARD Enable
"M17.2"	M 17.2	BOOL	// Loader BACKWARD Enable
"M22.6"	M 22.6	BOOL	// Automatic Clamp OPEN One-Shot
"M22.7"	M 22.7	BOOL	// Automatic Clamp OPEN One-Shot
"M23.0"	M 23.0	BOOL	// Automatic Clamp CLOSE One-Shot
"M23.1"	M 23.1	BOOL	// Automatic Clamp CLOSE One-Shot
"M30.1"	M 30.1	BOOL	// Loader in stand by zone
"Cyclic OB"	OB 1	OB 1	// Cyclic OB program
"A0.0"	Q 0.0	BOOL	// Loader General Fault Lamp - 283H1
"A0.1"	Q 0.1	BOOL	// Alarms RESET Lamp - 274S3
"A0.2"	Q 0.2	BOOL	// Drives Alarms Lamp - 274S4
"A0.3"	Q 0.3	BOOL	// Spare
"A0.4"	Q 0.4	BOOL	// Spare
"A0.5"	Q 0.5	BOOL	// Spare
"A0.6"	Q 0.6	BOOL	// Spare
"A0.7"	Q 0.7	BOOL	// Spare
"A1.0"	Q 1.0	BOOL	// Loader in STAND-BY Signal to MAIN BOARD
"A1.1"	Q 1.1	BOOL	// Loader INSIDE CAGE Signal to MAIN BOARD
"A1.2"	Q 1.2	BOOL	// Loader CLAMP OPEN Signal to MAIN BOARD
"A1.3"	Q 1.3	BOOL	// Loader in PARKING Signal to MAIN BOARD
"A1.4"	Q 1.4	BOOL	// Spare
"A1.5"	Q 1.5	BOOL	// Spare
"A1.6"	Q 1.6	BOOL	// Spare
"A1.7"	Q 1.7	BOOL	// Spare
"A124.0"	Q 124.0	BOOL	// Loader Clamp OPEN Motor - 281K1
"A124.1"	Q 124.1	BOOL	// Loader Clamp CLOSE Motor - 281K2
"A124.2"	Q 124.2	BOOL	// Loader Translation Drive Run Forward
"A124.3"	Q 124.3	BOOL	// Loader Translation Drive Run Backward
"A124.4"	Q 124.4	BOOL	// Loader Translation Drive Slow-Down
"A124.5"	Q 124.5	BOOL	// Loader Translation Drive Spare
"A124.6"	Q 124.6	BOOL	// Loader Translation Motor Brakes - 281K7
"A124.7"	Q 124.7	BOOL	// Spare
"A125.0"	Q 125.0	BOOL	// Loader Translation Drives Contactor - 282K1
"A125.1"	Q 125.1	BOOL	// Loader Lifting / Lower Motors 1 & 2 Drive Run FORWARD
"A125.2"	Q 125.2	BOOL	// Loader Lifting / Lower Motors 1 & 2 Drive Run BACKWARD
"A125.3"	Q 125.3	BOOL	// Loader Lifting / Lower Motors 1 & 2 Drive SLOW-DOWN
"A125.4"	Q 125.4	BOOL	// Loader Lifting / Lower Motors 1 & 2 Drive COAST STOP  ?????????
"A125.5"	Q 125.5	BOOL	// Loader Lifting / Lower Motors 1 & 2 Electrical Brakes
"A125.6"	Q 125.6	BOOL	// Spare
"A125.7"	Q 125.7	BOOL	// Loader Lifting / Lower Motors 1 & 2 Contactor Drive Run
END_SYMBOL_TABLE

FUNCTION "Cage Function" : VOID	// FC 7
AUTHOR : Manzoni
VERSION : 0.1
BEGIN
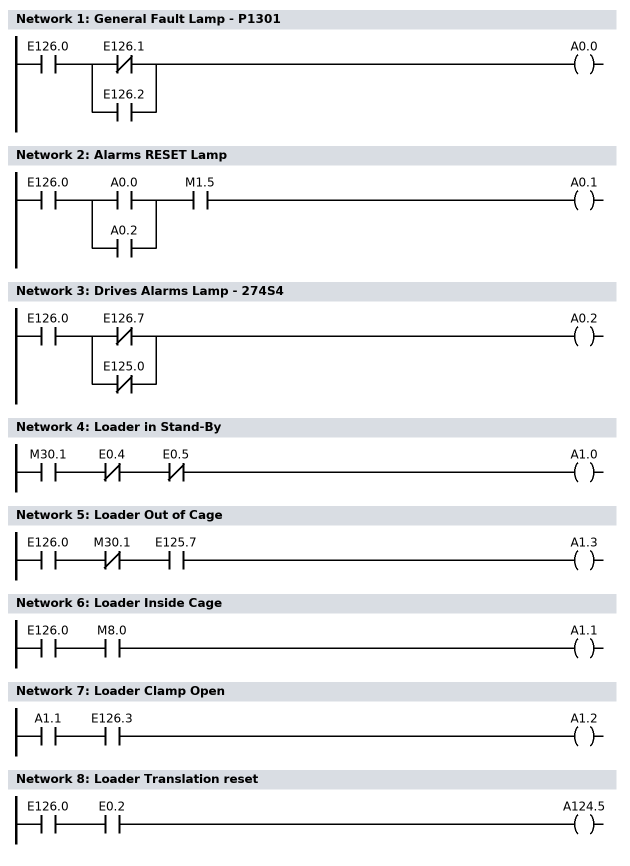
NETWORK
TITLE = General Fault Lamp - P1301
      A     "E126.0";
      A(;
      ON    "E126.1";
      O     "E126.2";
      );
      =     "A0.0";
NETWORK
TITLE = Alarms RESET Lamp
      A     "E126.0";
      A(;
      O     "A0.0";
      O     "A0.2";
      );
      A     "M1.5";
      =     "A0.1";
NETWORK
TITLE = Drives Alarms Lamp - 274S4
      A     "E126.0";
      A(;
      ON    "E126.7";
      ON    "E125.0";
      );
      =     "A0.2";
NETWORK
TITLE = Loader in Stand-By
      A     "M30.1";
      AN    "E0.4";
      AN    "E0.5";
      =     "A1.0";
NETWORK
TITLE = Loader Out of Cage
      A     "E126.0";
      AN    "M30.1";
      A     "E125.7";
      =     "A1.3";
NETWORK
TITLE = Loader Inside Cage
      A     "E126.0";
      A     "M8.0";
      =     "A1.1";
NETWORK
TITLE = Loader Clamp Open
      A     "A1.1";
      A     "E126.3";
      =     "A1.2";
NETWORK
TITLE = Loader Translation reset
//?????????????????
//?????????????????
//?????????????????
      A     "E126.0";
      A     "E0.2";
      =     "A124.5";
END_FUNCTION

FUNCTION "Translation Function" : VOID	// FC 8
AUTHOR : Manzoni
VERSION : 0.1
BEGIN
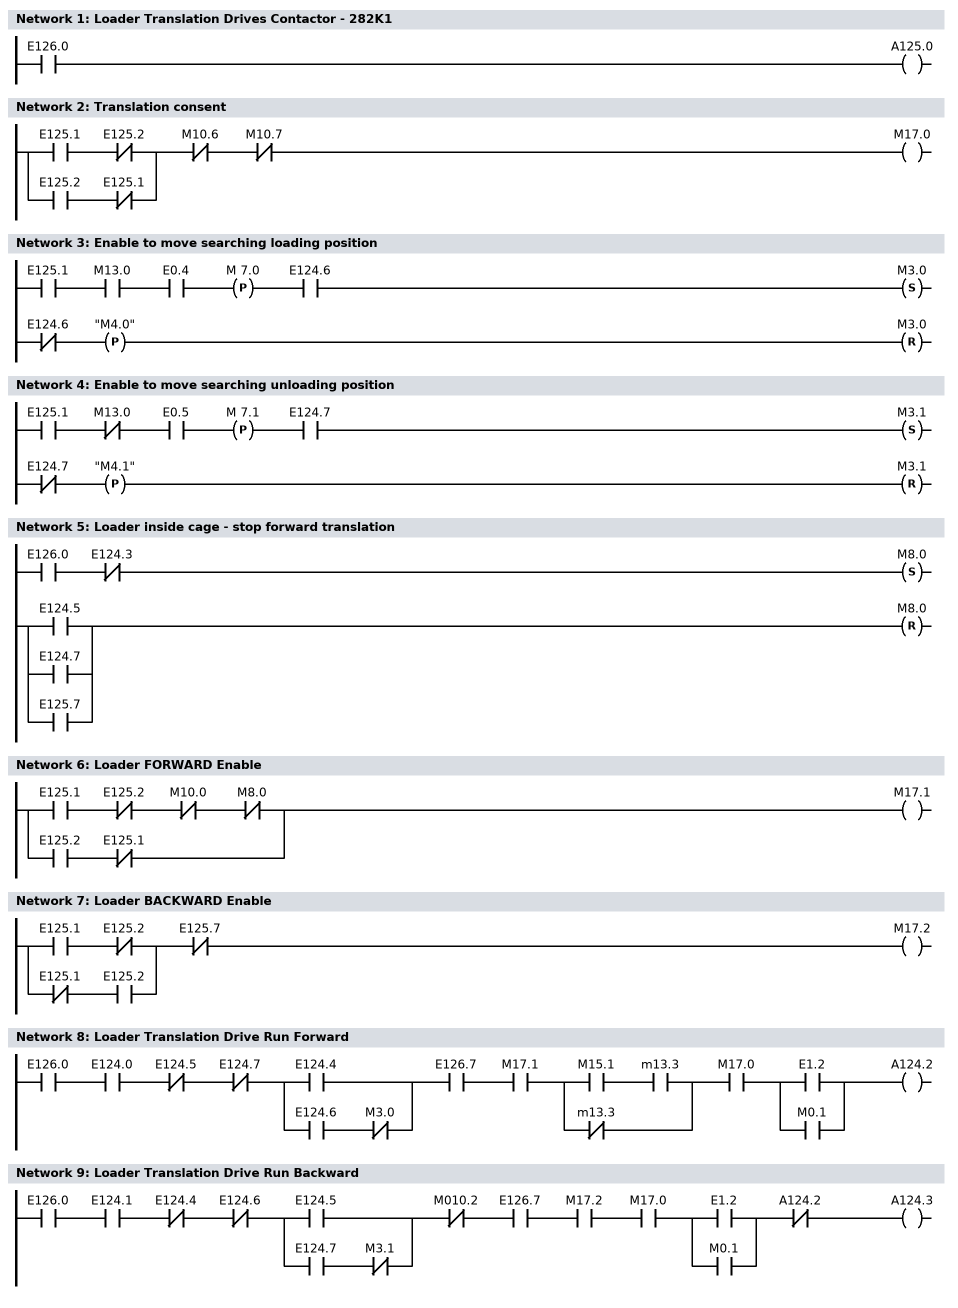
NETWORK
TITLE = Loader Translation Drives Contactor - 282K1
      A     "E126.0";
      =     "A125.0";
NETWORK
TITLE = Translation consent
      A(;
      A     "E125.1";
      AN    "E125.2";
      O;
      A     "E125.2";
      AN    "E125.1";
      );
      AN    "M10.6";
      AN    "M10.7";
      =     "M17.0";
NETWORK
TITLE = Enable to move searching loading position
      A     "E125.1";
      A     "M13.0";
      A     "E0.4";
      FP    M 7.0;
      A     "E124.6";
      S     "M3.0";
      AN    "E124.6";
      FP    "M4.0";
      R     "M3.0";
      NOP   0;
NETWORK
TITLE = Enable to move searching unloading position
      A     "E125.1";
      AN    "M13.0";
      A     "E0.5";
      FP    M 7.1;
      A     "E124.7";
      S     "M3.1";
      AN    "E124.7";
      FP    "M4.1";
      R     "M3.1";
      NOP   0;
NETWORK
TITLE = Loader inside cage - stop forward translation
      A     "E126.0";
      AN    "E124.3";
      S     "M8.0";
      A(;
      O     "E124.5";
      O     "E124.7";
      O     "E125.7";
      );
      R     "M8.0";
      NOP   0;
NETWORK
TITLE = Loader FORWARD Enable
      A     "E125.1";
      AN    "E125.2";
      AN    "M10.0";
      AN    "M8.0";
      O;
      A     "E125.2";
      AN    "E125.1";
      =     "M17.1";
NETWORK
TITLE = Loader BACKWARD Enable
      A(;
      A     "E125.1";
      AN    "E125.2";
      O;
      AN    "E125.1";
      A     "E125.2";
      );
      AN    "E125.7";
      =     "M17.2";
NETWORK
TITLE = Loader Translation Drive Run Forward
      A     "E126.0";
      A     "E124.0";
      AN    "E124.5";
      AN    "E124.7";
      A(;
      O     "E124.4";
      O;
      A     "E124.6";
      AN    "M3.0";
      );
      A     "E126.7";
      A     "M17.1";
      A(;
      A     "M15.1";
      A     "m13.3";
      ON    "m13.3";
      );
      A     "M17.0";
      A(;
      O     "E1.2";
      O     "M0.1";
      );
      =     "A124.2";
NETWORK
TITLE = Loader Translation Drive Run Backward
      A     "E126.0";
      A     "E124.1";
      AN    "E124.4";
      AN    "E124.6";
      A(;
      O     "E124.5";
      O;
      A     "E124.7";
      AN    "M3.1";
      );
      AN    "M010.2";
      A     "E126.7";
      A     "M17.2";
      A     "M17.0";
      A(;
      O     "E1.2";
      O     "M0.1";
      );
      AN    "A124.2";
      =     "A124.3";
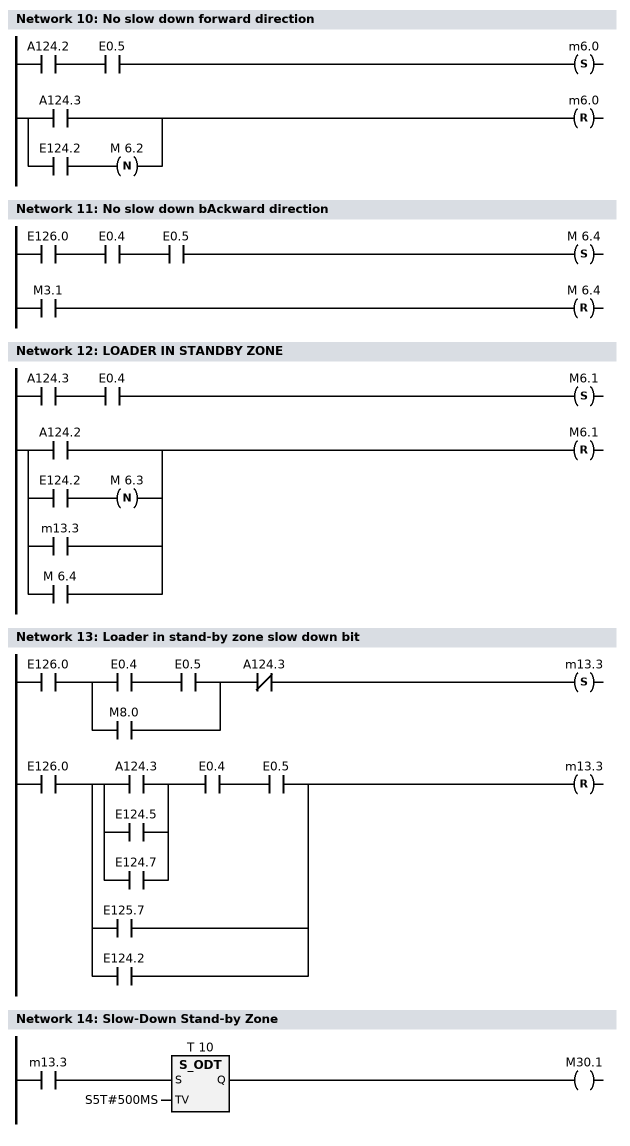
NETWORK
TITLE = No slow down forward direction
      A     "A124.2";
      A     "E0.5";
      S     "m6.0";
      A(;
      O     "A124.3";
      O(;
      A     "E124.2";
      FN    M 6.2;
      );
      );
      R     "m6.0";
      NOP   0;
NETWORK
TITLE = No slow down bAckward direction
      A     "E126.0";
      A     "E0.4";
      A     "E0.5";
      S     M 6.4;
      A     "M3.1";
      R     M 6.4;
      NOP   0;
NETWORK
TITLE = LOADER IN STANDBY ZONE
      A     "A124.3";
      A     "E0.4";
      S     "M6.1";
      A(;
      O     "A124.2";
      O(;
      A     "E124.2";
      FN    M 6.3;
      );
      O     "m13.3";
      O     M 6.4;
      );
      R     "M6.1";
      NOP   0;
NETWORK
TITLE = Loader in stand-by zone slow down bit
      A     "E126.0";
      A(;
      A     "E0.4";
      A     "E0.5";
      O     "M8.0";
      );
      AN    "A124.3";
      S     "m13.3";
      A     "E126.0";
      A(;
      A(;
      O     "A124.3";
      O     "E124.5";
      O     "E124.7";
      );
      A     "E0.4";
      A     "E0.5";
      O     "E125.7";
      O     "E124.2";
      );
      R     "m13.3";
      NOP   0;
NETWORK
TITLE = Slow-Down Stand-by Zone
      A     "m13.3";
      L     S5T#500MS;
      SD    T 10;
      NOP   0;
      NOP   0;
      NOP   0;
      A     T 10;
      =     "M30.1";
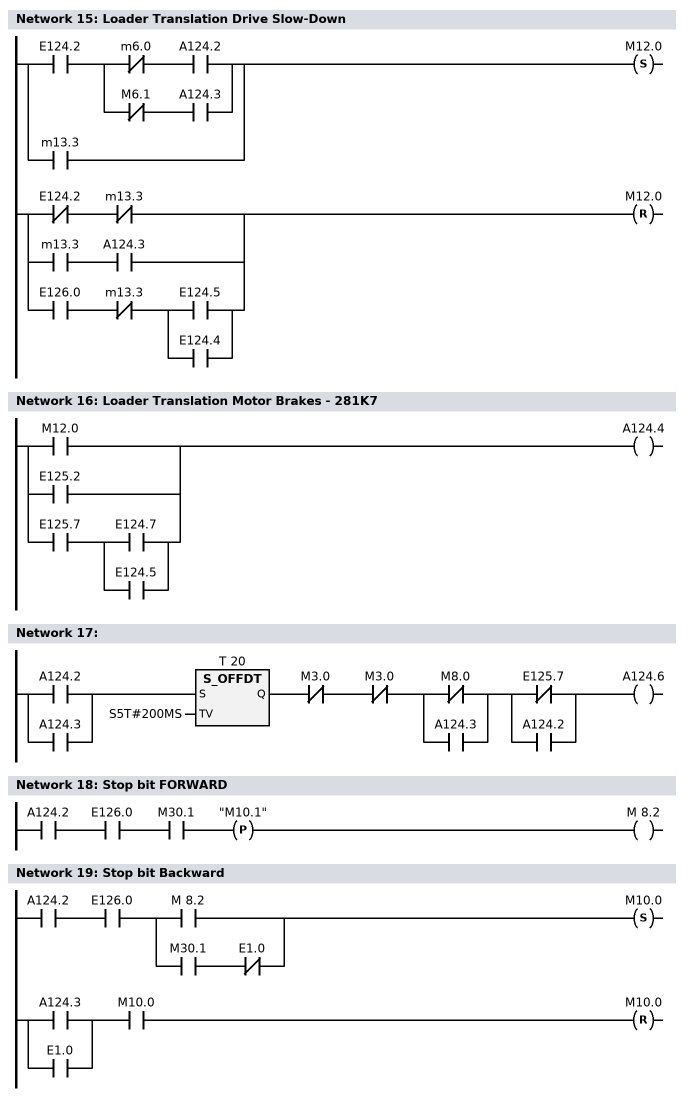
NETWORK
TITLE = Loader Translation Drive Slow-Down
      A(;
      A     "E124.2";
      A(;
      AN    "m6.0";
      A     "A124.2";
      O;
      AN    "M6.1";
      A     "A124.3";
      );
      O     "m13.3";
      );
      S     "M12.0";
      A(;
      AN    "E124.2";
      AN    "m13.3";
      O;
      A     "m13.3";
      A     "A124.3";
      O;
      A     "E126.0";
      AN    "m13.3";
      A(;
      O     "E124.5";
      O     "E124.4";
      );
      );
      R     "M12.0";
      NOP   0;
NETWORK
TITLE = Loader Translation Motor Brakes - 281K7
      O     "M12.0";
      O     "E125.2";
      O;
      A     "E125.7";
      A(;
      O     "E124.7";
      O     "E124.5";
      );
      =     "A124.4";
NETWORK
TITLE =
      A(;
      A(;
      O     "A124.2";
      O     "A124.3";
      );
      L     S5T#200MS;
      SF    T 20;
      NOP   0;
      NOP   0;
      NOP   0;
      A     T 20;
      );
      AN    "M3.0";
      AN    "M3.0";
      A(;
      ON    "M8.0";
      O     "A124.3";
      );
      A(;
      ON    "E125.7";
      O     "A124.2";
      );
      =     "A124.6";
NETWORK
TITLE = Stop bit FORWARD
      A     "A124.2";
      A     "E126.0";
      A     "M30.1";
      FP    "M10.1";
      =     M 8.2;
NETWORK
TITLE = Stop bit Backward
      A     "A124.2";
      A     "E126.0";
      A(;
      O     M 8.2;
      O;
      A     "M30.1";
      AN    "E1.0";
      );
      S     "M10.0";
      A(;
      O     "A124.3";
      O     "E1.0";
      );
      A     "M10.0";
      R     "M10.0";
      NOP   0;
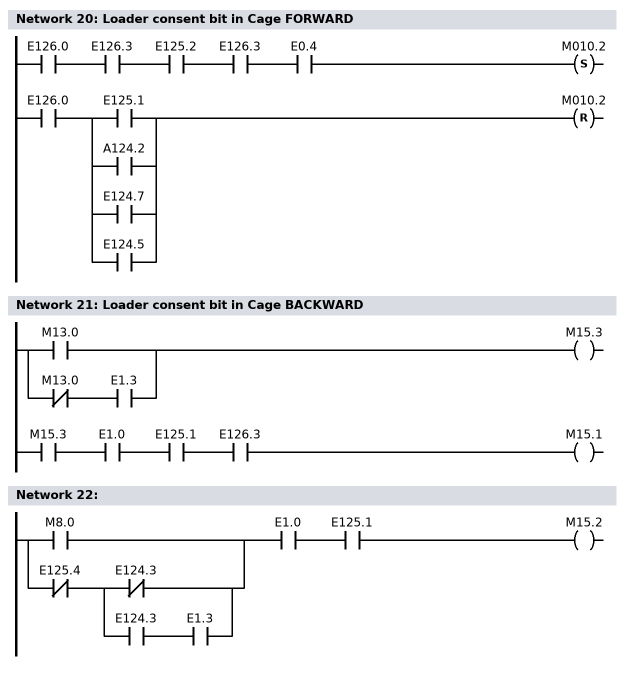
NETWORK
TITLE = Loader consent bit in Cage FORWARD
      A     "E126.0";
      A     "E126.3";
      A     "E125.2";
      A     "E126.3";
      A     "E0.4";
      S     "M010.2";
      A     "E126.0";
      A(;
      O     "E125.1";
      O     "A124.2";
      O     "E124.7";
      O     "E124.5";
      );
      R     "M010.2";
      NOP   0;
NETWORK
TITLE = Loader consent bit in Cage BACKWARD
      A(;
      O     "M13.0";
      O;
      AN    "M13.0";
      A     "E1.3";
      );
      =     "M15.3";
      A     "M15.3";
      A     "E1.0";
      A     "E125.1";
      A     "E126.3";
      =     "M15.1";
NETWORK
TITLE =
      A(;
      O     "M8.0";
      O;
      AN    "E125.4";
      A(;
      ON    "E124.3";
      O;
      A     "E124.3";
      A     "E1.3";
      );
      );
      A     "E1.0";
      A     "E125.1";
      =     "M15.2";
END_FUNCTION

FUNCTION "Clamp Function" : VOID	// FC 9
AUTHOR : Manzoni
VERSION : 0.1
BEGIN
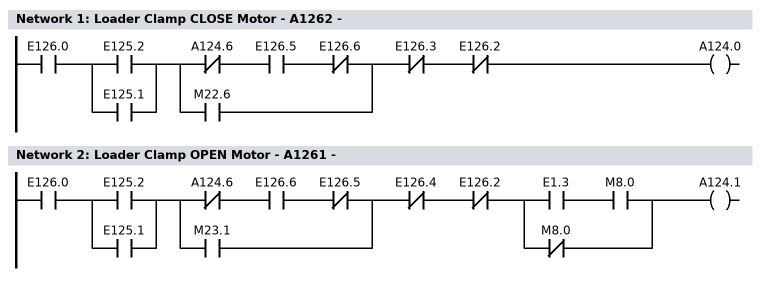
NETWORK
TITLE = Loader Clamp CLOSE Motor - A1262 -
      A     "E126.0";
      A(;
      O     "E125.2";
      O     "E125.1";
      );
      A(;
      AN    "A124.6";
      A     "E126.5";
      AN    "E126.6";
      O     "M22.6";
      );
      AN    "E126.3";
      AN    "E126.2";
      =     "A124.0";
NETWORK
TITLE = Loader Clamp OPEN Motor - A1261 -
      A     "E126.0";
      A(;
      O     "E125.2";
      O     "E125.1";
      );
      A(;
      AN    "A124.6";
      A     "E126.6";
      AN    "E126.5";
      O     "M23.1";
      );
      AN    "E126.4";
      AN    "E126.2";
      A(;
      A     "E1.3";
      A     "M8.0";
      ON    "M8.0";
      );
      =     "A124.1";
END_FUNCTION

FUNCTION "Rotation Function" : VOID	// FC 10
AUTHOR : Manzoni
VERSION : 0.1
BEGIN
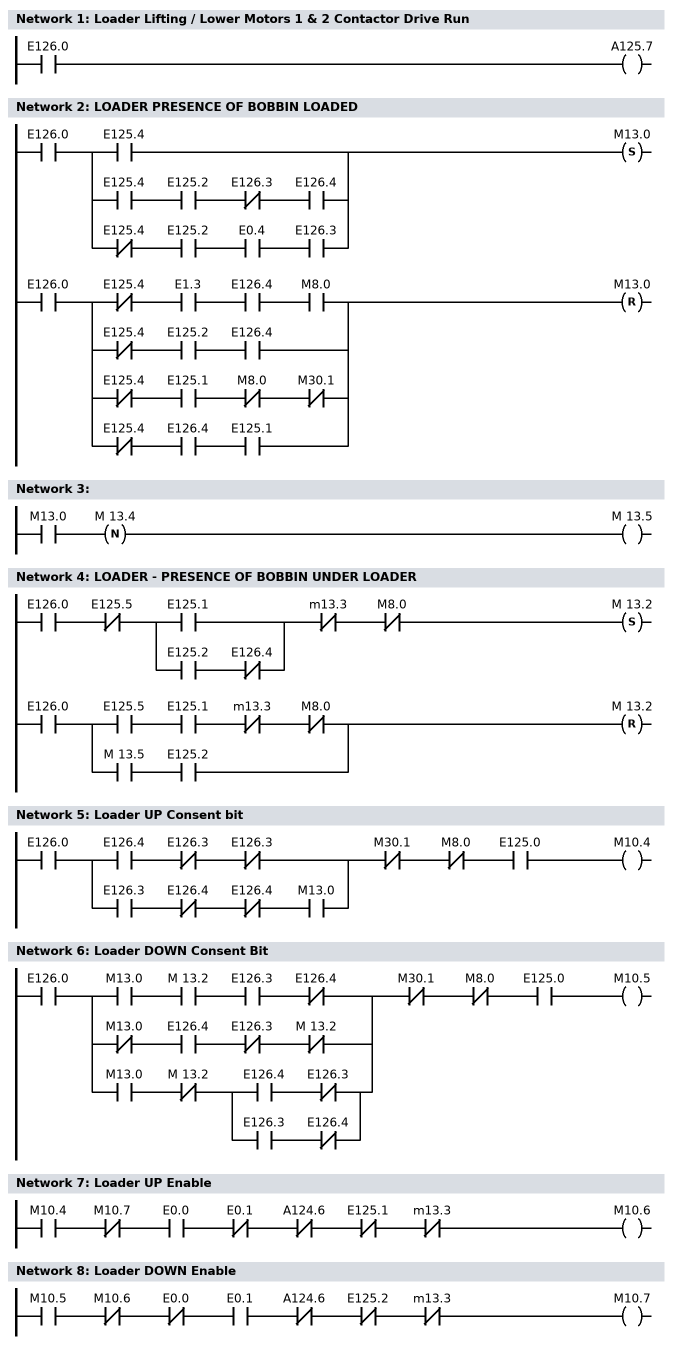
NETWORK
TITLE = Loader Lifting / Lower Motors 1 & 2 Contactor Drive Run
      A     "E126.0";
      =     "A125.7";
NETWORK
TITLE = LOADER PRESENCE OF BOBBIN LOADED
      A     "E126.0";
      A(;
      O     "E125.4";
      O;
      A     "E125.4";
      A     "E125.2";
      AN    "E126.3";
      A     "E126.4";
      O;
      AN    "E125.4";
      A     "E125.2";
      A     "E0.4";
      A     "E126.3";
      );
      S     "M13.0";
      A     "E126.0";
      A(;
      AN    "E125.4";
      A     "E1.3";
      A     "E126.4";
      A     "M8.0";
      O;
      AN    "E125.4";
      A     "E125.2";
      A     "E126.4";
      O;
      AN    "E125.4";
      A     "E125.1";
      AN    "M8.0";
      AN    "M30.1";
      O;
      AN    "E125.4";
      A     "E126.4";
      A     "E125.1";
      );
      R     "M13.0";
      NOP   0;
NETWORK
TITLE =
      A     "M13.0";
      FN    M 13.4;
      =     M 13.5;
NETWORK
TITLE = LOADER - PRESENCE OF BOBBIN UNDER LOADER
      A     "E126.0";
      AN    "E125.5";
      A(;
      O     "E125.1";
      O;
      A     "E125.2";
      AN    "E126.4";
      );
      AN    "m13.3";
      AN    "M8.0";
      S     M 13.2;
      A     "E126.0";
      A(;
      A     "E125.5";
      A     "E125.1";
      AN    "m13.3";
      AN    "M8.0";
      O;
      A     M 13.5;
      A     "E125.2";
      );
      R     M 13.2;
      NOP   0;
NETWORK
TITLE = Loader UP Consent bit
      A     "E126.0";
      A(;
      A     "E126.4";
      AN    "E126.3";
      AN    "E126.3";
      O;
      A     "E126.3";
      AN    "E126.4";
      AN    "E126.4";
      A     "M13.0";
      );
      AN    "M30.1";
      AN    "M8.0";
      A     "E125.0";
      =     "M10.4";
NETWORK
TITLE = Loader DOWN Consent Bit
      A     "E126.0";
      A(;
      A     "M13.0";
      A     M 13.2;
      A     "E126.3";
      AN    "E126.4";
      O;
      AN    "M13.0";
      A     "E126.4";
      AN    "E126.3";
      AN    M 13.2;
      O;
      A     "M13.0";
      AN    M 13.2;
      A(;
      A     "E126.4";
      AN    "E126.3";
      O;
      A     "E126.3";
      AN    "E126.4";
      );
      );
      AN    "M30.1";
      AN    "M8.0";
      A     "E125.0";
      =     "M10.5";
NETWORK
TITLE = Loader UP Enable
      A     "M10.4";
      AN    "M10.7";
      A     "E0.0";
      AN    "E0.1";
      AN    "A124.6";
      AN    "E125.1";
      AN    "m13.3";
      =     "M10.6";
NETWORK
TITLE = Loader DOWN Enable
      A     "M10.5";
      AN    "M10.6";
      AN    "E0.0";
      A     "E0.1";
      AN    "A124.6";
      AN    "E125.2";
      AN    "m13.3";
      =     "M10.7";
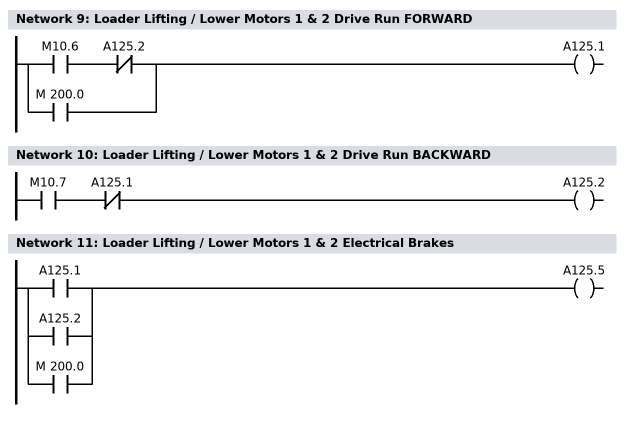
NETWORK
TITLE = Loader Lifting / Lower Motors 1 & 2 Drive Run FORWARD
      A     "M10.6";
      AN    "A125.2";
      O     M 200.0;
      =     "A125.1";
NETWORK
TITLE = Loader Lifting / Lower Motors 1 & 2 Drive Run BACKWARD
      A     "M10.7";
      AN    "A125.1";
      =     "A125.2";
NETWORK
TITLE = Loader Lifting / Lower Motors 1 & 2 Electrical Brakes
      O     "A125.1";
      O     "A125.2";
      O     M 200.0;
      =     "A125.5";
END_FUNCTION

ORGANIZATION_BLOCK "Cyclic OB"	// OB 1
AUTHOR : Manzoni
VERSION : 0.1
VAR_TEMP
  TEMP0 : BYTE ;
  TEMP1 : BYTE ;
  TEMP2 : BYTE ;
  TEMP3 : BYTE ;
  TEMP4 : BYTE ;
  TEMP5 : BYTE ;
  TEMP6 : INT ;
  TEMP7 : INT ;
  TEMP8 : INT ;
  TEMP9 : DATE_AND_TIME ;
END_VAR
BEGIN
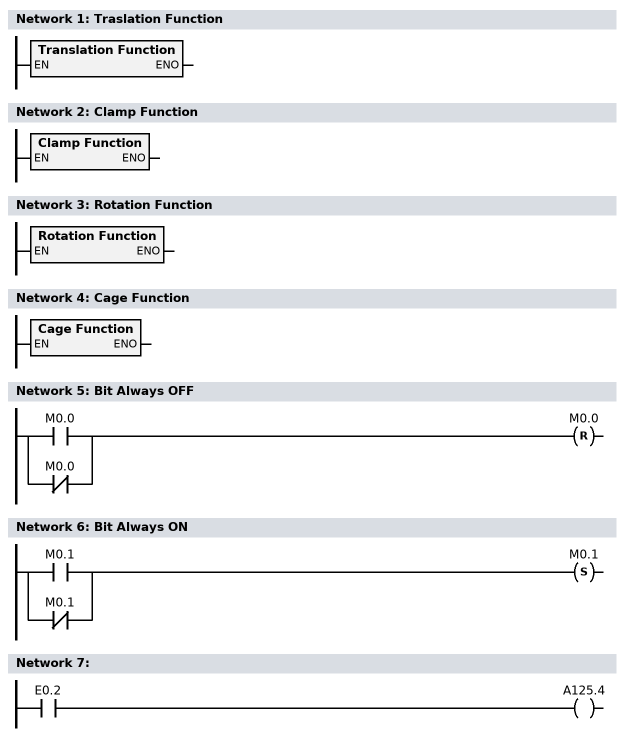
NETWORK
TITLE = Traslation Function
      CALL  "Translation Function";
      NOP   0;
NETWORK
TITLE = Clamp Function
      CALL  "Clamp Function";
      NOP   0;
NETWORK
TITLE = Rotation Function
      CALL  "Rotation Function";
      NOP   0;
NETWORK
TITLE = Cage Function
      CALL  "Cage Function";
      NOP   0;
NETWORK
TITLE = Bit Always OFF
      O     "M0.0";
      ON    "M0.0";
      R     "M0.0";
NETWORK
TITLE = Bit Always ON
      O     "M0.1";
      ON    "M0.1";
      S     "M0.1";
NETWORK
TITLE =
      A     "E0.2";
      =     "A125.4";
END_ORGANIZATION_BLOCK
